{attribute 'GeneratedUsingTerminal: CU1123-0010-0016'}
{attribute addProperty BoxType "CU1123-0010-0016"}
{attribute addProperty Id "A_0003_CU1124_0000_0016A_0003_CU1124_0000_0016_743794C092"}
{attribute addProperty CRC "3805748817"}
{attribute addProperty Size "92"}
TYPE A_0002_CU1123_0010_0016_E2D71E51 EXTENDS CU1123_1FC0878B :
STRUCT
	{attribute addProperty Name "A_0003_CU1124_0000_0016"}
	{attribute addProperty PreviousPort "A_0002(CU1123-0010-0016) : D"}
	A_0003_CU1124_0000_0016 : A_0003_CU1124_0000_0016_743794C0;
END_STRUCT
END_TYPE

(* stored: Version 1.2.0.0, ProductVersion 3.1.4024.9
   DUT A_0002_CU1123_0010_0016_E2D71E51: Id {7d22c1a5-49d5-4da7-9ea1-db188bcd3093} *)
